TYPE ST_TurntableMotionConfig :
STRUCT
    fVelocity : LREAL;
    fAcceleration : LREAL;
    fDeceleration : LREAL;
    fPositionTolerance : LREAL;
    tMoveTimeout : TIME;
END_STRUCT
END_TYPE

(* stored: Version 1.1.0.1, ProductVersion 3.1.4026.20
   DUT ST_TurntableMotionConfig: Id {a9500594-0156-4380-92f3-8b91658b6c65} *)
